# EPICS autosave request: dxp/tags/synApps_5_2/iocBoot/iocDXP2X/auto_settings.req
file "simple_mca_settings.req", P=dxp2X:, M=med:mca1
file "simple_mca_settings.req", P=dxp2X:, M=med:mca2
file "simple_mca_settings.req", P=dxp2X:, M=med:mca3
file "simple_mca_settings.req", P=dxp2X:, M=med:mca4
file "simple_mca_settings.req", P=dxp2X:, M=med:mca5
file "simple_mca_settings.req", P=dxp2X:, M=med:mca6
file "simple_mca_settings.req", P=dxp2X:, M=med:mca7
file "simple_mca_settings.req", P=dxp2X:, M=med:mca8
file "simple_mca_settings.req", P=dxp2X:, M=med:mca9
file "simple_mca_settings.req", P=dxp2X:, M=med:mca10
file "simple_mca_settings.req", P=dxp2X:, M=med:mca11
file "simple_mca_settings.req", P=dxp2X:, M=med:mca12
file "simple_mca_settings.req", P=dxp2X:, M=med:mca13
file "simple_mca_settings.req", P=dxp2X:, M=med:mca14
file "simple_mca_settings.req", P=dxp2X:, M=med:mca15
file "simple_mca_settings.req", P=dxp2X:, M=med:mca16
file "dxp_settings.req", P=dxp2X:, R=med:dxp1
file "dxp_settings.req", P=dxp2X:, R=med:dxp2
file "dxp_settings.req", P=dxp2X:, R=med:dxp3
file "dxp_settings.req", P=dxp2X:, R=med:dxp4
file "dxp_settings.req", P=dxp2X:, R=med:dxp5
file "dxp_settings.req", P=dxp2X:, R=med:dxp6
file "dxp_settings.req", P=dxp2X:, R=med:dxp7
file "dxp_settings.req", P=dxp2X:, R=med:dxp8
file "dxp_settings.req", P=dxp2X:, R=med:dxp9
file "dxp_settings.req", P=dxp2X:, R=med:dxp10
file "dxp_settings.req", P=dxp2X:, R=med:dxp11
file "dxp_settings.req", P=dxp2X:, R=med:dxp12
file "dxp_settings.req", P=dxp2X:, R=med:dxp13
file "dxp_settings.req", P=dxp2X:, R=med:dxp14
file "dxp_settings.req", P=dxp2X:, R=med:dxp15
file "dxp_settings.req", P=dxp2X:, R=med:dxp16
